FUNCTION_BLOCK E_RS (* Basic Function Block Type *)
  (* Standard: 61499-2 *)
  (* Version 0.0, 9/9/2026, lizar, Schneider Electric, Template *)
  PACKAGE Main;
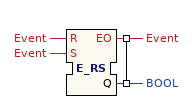
  EVENT_INPUT
    R; (* Initialization Request *)
    S; (* Normal Execution Request *)
  END_EVENT
  EVENT_OUTPUT
    EO WITH Q; (* Initialization Confirm *)
  END_EVENT
  VAR_OUTPUT
    Q : BOOL; (* Output event qualifier *)
  END_VAR
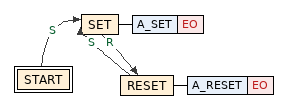
  EC_STATES
    START; (* Initial State *)
    SET : A_SET -> EO; (* Initialization *)
    RESET : A_RESET -> EO; (* Normal execution *)
  END_STATES
  EC_TRANSITIONS
    START TO SET := S;
    SET TO RESET := R;
    RESET TO SET := S;
  END_TRANSITIONS
  ALGORITHM A_SET IN ST:
Q:=1;
  END_ALGORITHM
  ALGORITHM A_RESET IN ST:
Q:=0;
  END_ALGORITHM
END_FUNCTION_BLOCK
